PROGRAM P_Modbus_RTU
VAR
	(*********************RTU******************************)
	master:ARRAY[1..2] OF    ModbusRtuMaster_KL6x22B;
    start:ARRAY[1..2] OF  BOOL:=[TRUE];
	step:ARRAY[1..2] OF  INT;
	
	com1_station:ARRAY[1..5] OF stRtu;
	
	tab_vac_measure	:ARRAY[1..2] OF WORD;//负压表值
	tab_vac_set		:ARRAY[1..2] OF WORD;//负压表值
	sub_pressure_measure	: LREAL;//sub测量正压
	sub_pressure_set		: LREAL;//sun正压设定值
	sub_vac_c_measure		: LREAL;//sub彩色负压值
	sub_vac_w_measure		: LREAL;//sub白色负压值
	sub_vac_c_set			: LREAL;//sub彩色负压设定值
	sub_vac_w_set			: LREAL;//sub白色负压设定值
	
	cycle_time:INT;
	count_time:INT:=5;
	i,j:INT;	
	error_trig :ARRAY[1..10] OF Tc2_Standard.R_TRIG;
	error_count:ARRAY[1..10] OF DINT;//错误计数
	station_error_trig:ARRAY[1..10] OF Tc2_Standard.R_TRIG;	
	station_error AT%Q*:ARRAY[1..10] OF BOOL;
	test_send:BOOL;
END_VAR

VAR PERSISTENT
	break_systime:ARRAY[1..10] OF DATE_AND_TIME;
END_VAR

ACT();

(******************************************台面负压****************************************************)
	(*原本接收10代表1KPA，但修改温控表，使10代表1*)
	(**********READ****负数=正数按位取反+1******************************)
	IF com1_station[1]._04readarray[1].15=0 THEN 
		GVL_API.stTableVacuum[1].vacuum_measured:=WORD_TO_LREAL(com1_station[1]._04readarray[1])/100;
	ELSE 
		GVL_API.stTableVacuum[1].vacuum_measured:=WORD_TO_LREAL(NOT(com1_station[1]._04readarray[1]-1))/100;
	END_IF
	(***************台面负压****write****)	
	com1_station[1]._06writesinglearray[1]:=NOT (LREAL_TO_WORD(GVL_API.stTableVacuum[1].setpoint*100))+1;///负数，反吗+1
	(***************台面负压****writPID*)
	IF 	GVL_API.stTableVacuum[1].ctrlP >0 THEN 	//P 不能为0
		com1_station[1]._06writesinglearray_PID[2]:=LREAL_TO_WORD(GVL_API.stTableVacuum[1].ctrlP*10);//制冷端P
	ELSE 
		com1_station[1]._06writesinglearray_PID[2]:=LREAL_TO_WORD(10*10);//制冷端P
	END_IF
		com1_station[1]._06writesinglearray_PID[4]:=LREAL_TO_WORD(GVL_API.stTableVacuum[1].ctrlI);
		com1_station[1]._06writesinglearray_PID[6]:=LREAL_TO_WORD(GVL_API.stTableVacuum[1].ctrlD);
	
		
(***************温湿度****************)
		gvl.humidity_measured:=	WORD_TO_LREAL(com1_station[3]._03readarray[1])/10;
		IF com1_station[3]._03readarray[1].15=0 THEN 
			gvl.temp_measured:=WORD_TO_LREAL(com1_station[3]._03readarray[2])/10;
		ELSIF com1_station[3]._03readarray[1].15=1 THEN
			gvl.temp_measured:= WORD_TO_LREAL(NOT(com1_station[3]._03readarray[2]-1))/10;
		END_IF
		
		
		
(**************二级墨盒正负压****************
	(**********SUB VAC 正压**************)
	sub_pressure_measure:=  WORD_TO_LREAL( com1_station[4]._03readarray[1])/1000;   //当前值
	
	com1_station[4]._03writearray[1]:=LREAL_TO_WORD(sub_pressure_set*1000);//正压设定
	com1_station[4]._03writearray[4]:=1;//正压自启动
	com1_station[4]._03writearray[4]:=12;//正压电机速度
	
	(**********SUB VAC 负压**************)
	sub_vac_c_measure:=WORD_TO_LREAL(com1_station[5]._03readarray[1])/1000;
	sub_vac_w_measure:=WORD_TO_LREAL(com1_station[5]._03readarray[2])/1000;
	
	com1_station[5]._03writearray[1]:=LREAL_TO_WORD(sub_vac_c_set*1000);
	com1_station[5]._03writearray[2]:=LREAL_TO_WORD(sub_vac_w_set*1000);
	com1_station[5]._03writearray[3]:=3;
	com1_station[5]._03writearray[4]:=3;
*)

ACTION ACT:
CASE step[1] OF 
0: //初始状态
		IF start[1] THEN
			step[1]:=10;
			cycle_time:=0;
		END_IF	
10://站1 04口读操作  真空吸附			
			IF cycle_time>=count_time THEN 
				cycle_time:=0;	
				FOR j:=1 TO 10 DO 
					error_count[j]:=0;
				END_FOR		
			END_IF
						
			master[1].ReadInputRegs(
				UnitID:= 1, 
				Quantity:=4, 
				MBAddr:= 16#03E8, 
				cbLength:= SIZEOF(com1_station[1]._04readarray), 
				pMemoryAddr:= ADR(com1_station[1]._04readarray), 
				Execute:= TRUE, 
				Timeout:= T#200MS);	
											
				IF NOT master[1].BUSY  THEN
					master[1].ReadRegs(Execute:= FALSE, );
					cycle_time:=cycle_time+1;
					step[1]:=20;									
				END_IF
				
				station_error_trig[1](CLK:=master[1].error , Q=> );	
				IF station_error_trig[1].Q THEN 
					error_count[1]:=error_count[1]+1;
				END_IF
20://站1 06口写操作	,设定负压	
			master[1].WriteSingleRegister(
				UnitID:= 1, 
				Quantity:=1, 
				MBAddr:= 0, 
				cbLength:= 2, 
				pMemoryAddr:= ADR(com1_station[1]._06writesinglearray[1]), 
				Execute:= TRUE, 
				Timeout:= T#200MS, 
				BUSY=> , 
				Error=> , 
				ErrorId=> , 
				cbRead=> );			
						
				IF NOT master[1].BUSY  THEN
					master[1].ReadRegs(Execute:= FALSE, );
					step[1]:=21;									
				END_IF
				
				station_error_trig[1](CLK:=master[1].error , Q=> );	
				IF station_error_trig[1].Q THEN 
					error_count[1]:=error_count[1]+1;
				END_IF
21://站1 06口写操作	,设定PID
			master[1].WriteRegs(
				UnitID:= 1, 
				Quantity:=SIZEOF(com1_station[1]._06writesinglearray_PID)/2, 
				MBAddr:= 16#0065, 
				cbLength:= SIZEOF(com1_station[1]._06writesinglearray_PID), 
				pMemoryAddr:= ADR(com1_station[1]._06writesinglearray_PID), 
				Execute:= TRUE, 
				Timeout:= T#200MS, 
				BUSY=> , 
				Error=> , 
				ErrorId=> , 
				cbRead=> );	
				
				
				station_error_trig[1](CLK:=master[1].error , Q=> );	
				IF station_error_trig[1].Q THEN 
					error_count[1]:=error_count[1]+1;
				END_IF	
				IF cycle_time=count_time AND error_count[1]>=2 THEN 
					station_error[1]:=TRUE;
				END_IF

				IF NOT master[1].BUSY  THEN
					master[1].ReadRegs(Execute:= FALSE );
					step[1]:=50;											              		
				END_IF	
(*3://站2 04口读操作
			master[1].ReadInputRegs(
				UnitID:= 2, 
				Quantity:=4, 
				MBAddr:= 16#03E8, 
				cbLength:= SIZEOF(com1_station[2]._04readarray), 
				pMemoryAddr:= ADR(com1_station[2]._04readarray), 
				Execute:= TRUE, 
				Timeout:= T#200MS, 
				 );	
					          
				station_error_trig[2](CLK:=master[1].error , Q=> );	
				IF station_error_trig[2].Q THEN 
					error_count_test[2]:=error_count_test[2]+1;
				END_IF	 
				IF cycle_time=count_time AND error_count_test[2]>=2 THEN 
					station_error[2]:=TRUE;
				END_IF

	
				IF NOT master[1].BUSY  THEN
					master[1].ReadRegs(Execute:= FALSE, );
					IF NOT station_error[2] THEN 
						step[1]:=4;									
					ELSIF station_error[2] THEN 
						step[1]:=5;	
					END_IF		              		
				END_IF					 	
4://站2 06口写操作			
			master[1].WriteSingleRegister(
				UnitID:= 2, 
				Quantity:=1, 
				MBAddr:= 0, 
				cbLength:= SIZEOF(com1_station[2]._06writesinglearray[1]), 
				pMemoryAddr:= ADR(com1_station[2]._06writesinglearray[1]), 
				Execute:= TRUE, 
				Timeout:= T#200MS, 
				BUSY=> , 
				Error=> , 
				ErrorId=> , 
				cbRead=> );			
				
			
				station_error_trig[2](CLK:=master[1].error , Q=> );	
				IF station_error_trig[2].Q THEN 
					error_count_test[2]:=error_count_test[2]+1;
				END_IF	
				IF cycle_time=count_time AND error_count_test[2]>=2 THEN 
					station_error[2]:=TRUE;
				END_IF

				IF NOT master[1].BUSY  THEN
					master[1].ReadRegs(Execute:= FALSE, );					
					IF NOT station_error[2] THEN 
						step[1]:=5;									
					ELSIF station_error[2] THEN 
						step[1]:=5;	
					END_IF		              		
				END_IF		
*)				 	
50://站3温湿度 03读
			master[1].ReadRegs(
				UnitID:= 3, 
				Quantity:=2, 
				MBAddr:= 0, 
				cbLength:= SIZEOF(com1_station[3]._03readarray), 
				pMemoryAddr:= ADR(com1_station[3]._03readarray), 
				Execute:= TRUE, 
				Timeout:= T#200MS, 
				 );	
							     
				station_error_trig[3](CLK:=master[1].error , Q=> );	
				IF station_error_trig[3].Q THEN 
					error_count[3]:=error_count[3]+1;
				END_IF
				IF cycle_time=count_time AND error_count[3]>=2 THEN 
					station_error[3]:=TRUE;
				END_IF
								
				IF NOT master[1].BUSY  THEN
					master[1].ReadRegs(Execute:= FALSE, );										
					step[1]:=10;															              		
				END_IF
				
(*							
6://站4，正压板 03口读操作  当前压墨板正压传感器值，单位0.1kPa	
	     master[1].ReadRegs(
				UnitID:= 16#48, 
				Quantity:=7, 
				MBAddr:= 0, 
				cbLength:= SIZEOF(com1_station[4]._03readarray), 
				pMemoryAddr:= ADR(com1_station[4]._03readarray), 
				Execute:= TRUE, 
				Timeout:= T#200MS, 
				 );	
							
				station_error_trig[4](CLK:=master[1].error , Q=> );	
				IF station_error_trig[4].Q THEN 
					error_count_test[4]:=error_count_test[4]+1;
				END_IF		
			
				IF cycle_time=count_time AND error_count_test[4]>=2 THEN 
					station_error[4]:=TRUE;
				END_IF
				
				IF NOT master[1].BUSY  THEN
					master[1].ReadRegs(Execute:= FALSE, );					
					IF NOT station_error[4] THEN 
						step[1]:=7;									
					ELSIF station_error[4] THEN 
						step[1]:=8;	
					END_IF		              		
				END_IF						     					
7://站4，正压板 03口写操作 设定的压墨值，单位0.1kPa，绝对值。
		master[1].WriteRegs(
				UnitID:= 16#48, 
				Quantity:=6, 
				MBAddr:= 1, 
				cbLength:= SIZEOF(com1_station[4]._03writearray), 
				pMemoryAddr:= ADR(com1_station[4]._03writearray), 
				Execute:= TRUE, 
				Timeout:= T#200MS, 
				BUSY=> , 
				Error=> , 
				ErrorId=> , 
				cbRead=> );			
						
				station_error_trig[4](CLK:=master[1].error , Q=> );	
				IF station_error_trig[4].Q THEN 
					error_count_test[4]:=error_count_test[4]+1;
				END_IF	
				IF cycle_time=count_time AND error_count_test[4]>=2 THEN 
					station_error[4]:=TRUE;
				END_IF
				
				IF NOT master[1].BUSY  AND NOT station_error[4]THEN
					master[1].ReadRegs(Execute:= FALSE, );	
					step[1]:=8;
				ELSIF station_error[4] THEN 
					step[1]:=8;
				END_IF
				IF NOT master[1].BUSY  THEN
					master[1].ReadRegs(Execute:= FALSE, );					
					IF NOT station_error[4] THEN 
						step[1]:=8;									
					ELSIF station_error[4] THEN 
						step[1]:=8;	
					END_IF		              		
				END_IF					     				
8://zhan 5负压板 03口读操作
		master[1].ReadRegs(
				UnitID:= 16#1D, 
				Quantity:=8, 
				MBAddr:= 0, 
				cbLength:= SIZEOF(com1_station[5]._03readarray), 
				pMemoryAddr:= ADR(com1_station[5]._03readarray), 
				Execute:= TRUE, 
				Timeout:= T#200MS, 
				 );	
				
				station_error_trig[5](CLK:=master[1].error , Q=> );	
				IF station_error_trig[5].Q THEN 
					error_count_test[5]:=error_count_test[5]+1;
				END_IF	

				IF cycle_time=count_time AND error_count_test[5]>=2 THEN 
					station_error[5]:=TRUE;
				END_IF
				
				IF NOT master[1].BUSY  THEN
					master[1].ReadRegs(Execute:= FALSE, );					
					IF NOT station_error[5] THEN 
						step[1]:=9;									
					ELSIF station_error[5] THEN 
						step[1]:=1;	
					END_IF		              		
				END_IF							     
9://zhan 5,负压板 03口写	
		master[1].WriteRegs(
				UnitID:= 16#1D, 
				Quantity:=4, 
				MBAddr:= 2, 
				cbLength:= SIZEOF(com1_station[5]._03writearray), 
				pMemoryAddr:= ADR(com1_station[5]._03writearray), 
				Execute:= TRUE, 
				Timeout:= T#200MS, 
				BUSY=> , 
				Error=> , 
				ErrorId=> , 
				cbRead=> );			
				
		
				station_error_trig[5](CLK:=master[1].error , Q=> );	
				IF station_error_trig[5].Q THEN 
					error_count_test[5]:=error_count_test[5]+1;
				END_IF	
				
				IF cycle_time=count_time AND error_count_test[5]>=2 THEN 
					station_error[5]:=TRUE;
				END_IF
					
				IF NOT master[1].BUSY  THEN
					master[1].ReadRegs(Execute:= FALSE, );					
					IF NOT station_error[5] THEN 
						step[1]:=1;									
					ELSIF station_error[5] THEN 
						step[1]:=1;	
					END_IF		              		
				END_IF	
*)
END_CASE

IF GVL_API.stTableVacuum[1].Setoff (*OR GVL_API.stTableVacuum[2].Setoff*) THEN 
	station_error[1]:=FALSE;
	//station_error[2]:=FALSE;
END_IF
IF   GVL_API.stSystemEnvironment.Reset THEN 
	station_error[3]:=FALSE;
END_IF


FOR i:=1 TO 5 DO
 error_trig[i](CLK:=station_error[i] , Q=> );
	IF  error_trig[i].Q THEN 
		break_systime[i]:=systime.dttime;		
	END_IF
END_FOR
END_ACTION

END_PROGRAM

(* stored: Version 1.1.0.1, ProductVersion 3.1.4024.11
   POU P_Modbus_RTU: Id {69b12c10-67fd-4d9c-8cfe-ca4f157ddaa0}, SpecialFunc None
   Action ACT: Id {55d976e6-c45b-4e23-a100-16a0779c7add} *)
